FUNCTION IncIndex : INT
VAR_INPUT
	IDX:	INT;		// Index to be incremented
	IdxMIN:	INT;		// Min Value for index	
	IdxMAX:	INT;		// Max Value for index
END_VAR
VAR
END_VAR

IF IDX < IdxMAX THEN
	IncIndex := IDX + 1; 
ELSIF IDX = IdxMAX THEN
	IncIndex := IdxMIN;
ELSIF IDX < IdxMIN OR IDX > IdxMAX THEN
	 IncIndex := IdxMIN;
END_IF

END_FUNCTION

(* stored: Version 1.1.0.1, ProductVersion 3.1.4024.4
   POU IncIndex: Id {b01832d5-0bc7-4e64-a640-c1ca7a1a204c}, SpecialFunc None *)
